// TIA Portal project "HW_2200220OffsetBodu_V18_V19" (V19)

(* hardware
DEVICE "ET 200SP station_1"  ET 200SP-Station
   slot 0: "IO-R3"  Rack  6ES5 710-8MAx1
   slot 0: "A6"  IM 155-6 PN ST  6ES7 155-6AU01-0BN0  V4.2
   slot 1: "15A2"  DI 16x24VDC ST  6ES7 131-6BH01-0BA0  V0.0
      slot 1: "15A2"  DI 16x24VDC ST
   slot 2: "15A3"  DI 16x24VDC ST  6ES7 131-6BH01-0BA0  V0.0
      slot 1: "15A3"  DI 16x24VDC ST
   slot 3: "15A4"  DI 16x24VDC ST  6ES7 131-6BH01-0BA0  V0.0
      slot 1: "15A4"  DI 16x24VDC ST
   slot 4: "15A5"  DQ 16x24VDC/0.5A ST  6ES7 132-6BH01-0BA0  V0.0
      slot 1: "15A5"  DQ 16x24VDC/0.5A ST
   slot 5: "15A6"  DQ 16x24VDC/0.5A ST  6ES7 132-6BH01-0BA0  V0.0
      slot 1: "15A6"  DQ 16x24VDC/0.5A ST
   slot 6: "15A7"  DQ 16x24VDC/0.5A ST  6ES7 132-6BH01-0BA0  V0.0
      slot 1: "15A7"  DQ 16x24VDC/0.5A ST
   slot 7: "15A8"  DQ 16x24VDC/0.5A ST  6ES7 132-6BH01-0BA0  V0.0
      slot 1: "15A8"  DQ 16x24VDC/0.5A ST
   slot 8: "15A9"  AI 4xU/I 2-wire ST  6ES7 134-6HD00-0BA1  V1.1
      slot 1: "15A9"  AI 4xU/I 2-wire ST
   slot 9: "15A10"  AQ 4xU/I ST  6ES7 135-6HD00-0BA1  V1.1
      slot 1: "15A10"  AQ 4xU/I ST
   slot 15: "Server module_1"  Server module  6ES7 193-6PA00-0AA0  V1.0
      slot 1: "Server module_1"  Server module
   slot 127: "PROFINET BusAdapter CU"  BA 2xRJ45  6ES7 193-6AR00-0AA0  V0.0
      slot 1: "Port_1"  X1 P1 R  6ES7 193-6AR00-0AA0  V0.0
      slot 2: "Port_2"  X1 P2 R  6ES7 193-6AR00-0AA0  V0.0
DEVICE "GSD device_7"  GSD.Device.PN
   slot 0: "Rack"  Rack  V1.0
   slot 0: "VI-13"  CPX Rev 30  TN 197330  V4.2.30
      slot 0: "CPX Rev 30"  CPX Rev 30
      slot 1: "PN-IO Interface"  PN-IO Interface
         slot 1: "Port 1"  Port 1
         slot 2: "Port 2"  Port 2
   slot 1: "FB33 PNIO Module_1"  FB33 PNIO Module  TN 548755, CPX-FB33, Code F33
      slot 0: "FB33 PNIO Module"  FB33 PNIO Module
   slot 2: "MPA1S VMPA1-FB-EMS-8 [8DO]_1"  MPA1S VMPA1-FB-EMS-8 [8DO]  TN 533360, VMPA1-FB-EMS-8, Code A
      slot 0: "MPA1S VMPA1-FB-EMS-8 [8DO]"  MPA1S VMPA1-FB-EMS-8 [8DO]
   slot 3: "MPA1S VMPA1-FB-EMS-8 [8DO]_2"  MPA1S VMPA1-FB-EMS-8 [8DO]  TN 533360, VMPA1-FB-EMS-8, Code A
      slot 0: "MPA1S VMPA1-FB-EMS-8 [8DO]"  MPA1S VMPA1-FB-EMS-8 [8DO]
   slot 4: "MPA1S VMPA1-FB-EMS-8 [8DO]_3"  MPA1S VMPA1-FB-EMS-8 [8DO]  TN 533360, VMPA1-FB-EMS-8, Code A
      slot 0: "MPA1S VMPA1-FB-EMS-8 [8DO]"  MPA1S VMPA1-FB-EMS-8 [8DO]
   slot 5: "MPA1S VMPA1-FB-EMS-8 [8DO]_4"  MPA1S VMPA1-FB-EMS-8 [8DO]  TN 533360, VMPA1-FB-EMS-8, Code A
      slot 0: "MPA1S VMPA1-FB-EMS-8 [8DO]"  MPA1S VMPA1-FB-EMS-8 [8DO]
   slot 6: "MPA1S VMPA1-FB-EMS-8 [8DO]_5"  MPA1S VMPA1-FB-EMS-8 [8DO]  TN 533360, VMPA1-FB-EMS-8, Code A
      slot 0: "MPA1S VMPA1-FB-EMS-8 [8DO]"  MPA1S VMPA1-FB-EMS-8 [8DO]
   slot 7: "MPA1S VMPA1-FB-EMS-8 [8DO]_6"  MPA1S VMPA1-FB-EMS-8 [8DO]  TN 533360, VMPA1-FB-EMS-8, Code A
      slot 0: "MPA1S VMPA1-FB-EMS-8 [8DO]"  MPA1S VMPA1-FB-EMS-8 [8DO]
   slot 8: "MPA1S VMPA1-FB-EMS-8 [8DO]_7"  MPA1S VMPA1-FB-EMS-8 [8DO]  TN 533360, VMPA1-FB-EMS-8, Code A
      slot 0: "MPA1S VMPA1-FB-EMS-8 [8DO]"  MPA1S VMPA1-FB-EMS-8 [8DO]
   slot 9: "MPA1S VMPA1-FB-EMS-8 [8DO]_8"  MPA1S VMPA1-FB-EMS-8 [8DO]  TN 533360, VMPA1-FB-EMS-8, Code A
      slot 0: "MPA1S VMPA1-FB-EMS-8 [8DO]"  MPA1S VMPA1-FB-EMS-8 [8DO]
DEVICE "Connection Box_1"  SCALANCE X-Station
   slot 0: "Connection Box"  Rail
   slot 0: "ConBox"  Connection Box advanced  6AV2 125-2AE23-0AX0  V5.2
DEVICE "GSD device_3"  GSD.Device.PN
   slot 0: "Rack"  Rack  V1.0
   slot 0: "AxisLinear"  CMMT-AS V1  CMMT-AS-...-PN
      slot 0: "CMMT-AS V1"  CMMT-AS V1
      slot 1: "PN-IO Interface"  PN-IO Interface
         slot 1: "Port 1"  Port 1
         slot 2: "Port 2"  Port 2
      slot 1: "DO SERVO_1"  DO SERVO
         slot 0: "Module Access Point"  Module Access Point
   slot 2: "Siemens telegram 111, PZD-12/12"  Siemens telegram 111, PZD-12/12
DEVICE "ET 200AL station_1"  ET 200AL-Station
   slot 0: "Rack_0"  Rack
   slot 0: "52K1"  IM 157-1 PN  6ES7 157-1AB00-0AB0  V1.0
      slot 1: "ET-Con_1"  ET-Con IM Sub-Sender
      slot 1: "ET-Con_2"  ET-Con IM Sub-Sender
   slot 1: "Rack_1"  Rack  6ES714x-xxxxx-0AA0
   slot 2: "Rack_2"  Rack  6ES714x-xxxxx-0AA0
   slot 2: "53AB1"  DI 8x24VDC 8xM8  6ES7 141-5BF00-0BA0  V1.0
      slot 1: "53AB1"  DI 8x24VDC 8xM8  6ES7 141-5BF00-0BA0
      slot 2: "ET-Connection receiver"  ET-Con Sub-Receiver
   slot 3: "54AB2"  DI 8x24VDC 8xM8  6ES7 141-5BF00-0BA0  V1.0
      slot 1: "54AB2"  DI 8x24VDC 8xM8  6ES7 141-5BF00-0BA0
   slot 4: "55AB3"  DI 8x24VDC 8xM8  6ES7 141-5BF00-0BA0  V1.0
      slot 1: "55AB3"  DI 8x24VDC 8xM8  6ES7 141-5BF00-0BA0
   slot 5: "56AB4"  DI 8x24VDC 8xM8  6ES7 141-5BF00-0BA0  V1.0
      slot 1: "56AB4"  DI 8x24VDC 8xM8  6ES7 141-5BF00-0BA0
   slot 6: "57AB5"  DI 8x24VDC 8xM8  6ES7 141-5BF00-0BA0  V1.0
      slot 1: "57AB5"  DI 8x24VDC 8xM8  6ES7 141-5BF00-0BA0
   slot 19: "58AB6"  AI 4xU/I/RTD 4xM12  6ES7 144-5KD00-0BA0  V1.0
      slot 1: "58AB6"  AI 4xU/I/RTD 4xM12  6ES7 144-5KD00-0BA0
      slot 2: "ET-Connection receiver"  ET-Con Sub-Receiver
   slot 20: "59AB7"  DI 8x24VDC 8xM8  6ES7 141-5BF00-0BA0  V1.0
      slot 1: "59AB7"  DI 8x24VDC 8xM8  6ES7 141-5BF00-0BA0
   slot 21: "59aAB7"  DI 8x24VDC 8xM8  6ES7 141-5BF00-0BA0  V1.0
      slot 1: "59aAB7"  DI 8x24VDC 8xM8  6ES7 141-5BF00-0BA0
   slot 22: "60AB8"  DI 8x24VDC 8xM8  6ES7 141-5BF00-0BA0  V1.0
      slot 1: "60AB8"  DI 8x24VDC 8xM8  6ES7 141-5BF00-0BA0
   slot 23: "61AB9"  DI 8x24VDC 8xM8  6ES7 141-5BF00-0BA0  V1.0
      slot 1: "61AB9"  DI 8x24VDC 8xM8  6ES7 141-5BF00-0BA0
   slot 24: "62AB10"  DI 8x24VDC 8xM8  6ES7 141-5BF00-0BA0  V1.0
      slot 1: "62AB10"  DI 8x24VDC 8xM8  6ES7 141-5BF00-0BA0
DEVICE "CVIC II R2 A"  GSD.Device.PN
   slot 0: "Rack"  Rack  V1.0
   slot 0: "Bash"  RT  ABCC-PRT  V1.11
      slot 0: "RT"  RT
      slot 1: "Interface"  Interface
         slot 1: "Port 1"  Port 1
   slot 1: "Input 1 byte_1"  Input 1 byte  ABCC-PRT  V1.0
      slot 0: "Input 1 byte"  Input 1 byte
   slot 2: "Input 1 byte_2"  Input 1 byte  ABCC-PRT  V1.0
      slot 0: "Input 1 byte"  Input 1 byte
   slot 3: "Input 2 word_1"  Input 2 word  ABCC-PRT  V1.0
      slot 0: "Input 2 word"  Input 2 word
   slot 4: "Input 1 word_1"  Input 1 word  ABCC-PRT  V1.0
      slot 0: "Input 1 word"  Input 1 word
   slot 5: "Input 2 word_2"  Input 2 word  ABCC-PRT  V1.0
      slot 0: "Input 2 word"  Input 2 word
   slot 6: "Input 1 word_2"  Input 1 word  ABCC-PRT  V1.0
      slot 0: "Input 1 word"  Input 1 word
   slot 7: "Output 1 byte_1"  Output 1 byte  ABCC-PRT  V1.0
      slot 0: "Output 1 byte"  Output 1 byte
   slot 8: "Output 1 byte_2"  Output 1 byte  ABCC-PRT  V1.0
      slot 0: "Output 1 byte"  Output 1 byte
DEVICE "CVIC II R2 A_1"  GSD.Device.PN
   slot 0: "Rack"  Rack  V1.0
   slot 0: "AEBDown"  RT  ABCC-PRT  V1.11
      slot 0: "RT"  RT
      slot 1: "Interface"  Interface
         slot 1: "Port 1"  Port 1
   slot 1: "Input 1 byte_1"  Input 1 byte  ABCC-PRT  V1.0
      slot 0: "Input 1 byte"  Input 1 byte
   slot 2: "Input 1 byte_2"  Input 1 byte  ABCC-PRT  V1.0
      slot 0: "Input 1 byte"  Input 1 byte
   slot 3: "Input 2 word_1"  Input 2 word  ABCC-PRT  V1.0
      slot 0: "Input 2 word"  Input 2 word
   slot 4: "Input 1 word_1"  Input 1 word  ABCC-PRT  V1.0
      slot 0: "Input 1 word"  Input 1 word
   slot 5: "Input 2 word_2"  Input 2 word  ABCC-PRT  V1.0
      slot 0: "Input 2 word"  Input 2 word
   slot 6: "Input 1 word_2"  Input 1 word  ABCC-PRT  V1.0
      slot 0: "Input 1 word"  Input 1 word
   slot 7: "Output 1 byte_1"  Output 1 byte  ABCC-PRT  V1.0
      slot 0: "Output 1 byte"  Output 1 byte
   slot 8: "Output 1 byte_2"  Output 1 byte  ABCC-PRT  V1.0
      slot 0: "Output 1 byte"  Output 1 byte
DEVICE "CVIC II R2 A_2"  GSD.Device.PN
   slot 0: "Rack"  Rack  V1.0
   slot 0: "AEBUp"  RT  ABCC-PRT  V1.11
      slot 0: "RT"  RT
      slot 1: "Interface"  Interface
         slot 1: "Port 1"  Port 1
   slot 1: "Input 1 byte_1"  Input 1 byte  ABCC-PRT  V1.0
      slot 0: "Input 1 byte"  Input 1 byte
   slot 2: "Input 1 byte_2"  Input 1 byte  ABCC-PRT  V1.0
      slot 0: "Input 1 byte"  Input 1 byte
   slot 3: "Input 2 word_1"  Input 2 word  ABCC-PRT  V1.0
      slot 0: "Input 2 word"  Input 2 word
   slot 4: "Input 1 word_1"  Input 1 word  ABCC-PRT  V1.0
      slot 0: "Input 1 word"  Input 1 word
   slot 5: "Input 2 word_2"  Input 2 word  ABCC-PRT  V1.0
      slot 0: "Input 2 word"  Input 2 word
   slot 6: "Input 1 word_2"  Input 1 word  ABCC-PRT  V1.0
      slot 0: "Input 1 word"  Input 1 word
   slot 7: "Output 1 byte_1"  Output 1 byte  ABCC-PRT  V1.0
      slot 0: "Output 1 byte"  Output 1 byte
   slot 8: "Output 1 byte_2"  Output 1 byte  ABCC-PRT  V1.0
      slot 0: "Output 1 byte"  Output 1 byte
DEVICE "CVIC II R2 A_3"  GSD.Device.PN
   slot 0: "Rack"  Rack  V1.0
   slot 0: "AETDown"  RT  ABCC-PRT  V1.11
      slot 0: "RT"  RT
      slot 1: "Interface"  Interface
         slot 1: "Port 1"  Port 1
   slot 1: "Input 1 byte_1"  Input 1 byte  ABCC-PRT  V1.0
      slot 0: "Input 1 byte"  Input 1 byte
   slot 2: "Input 1 byte_2"  Input 1 byte  ABCC-PRT  V1.0
      slot 0: "Input 1 byte"  Input 1 byte
   slot 3: "Input 2 word_1"  Input 2 word  ABCC-PRT  V1.0
      slot 0: "Input 2 word"  Input 2 word
   slot 4: "Input 1 word_1"  Input 1 word  ABCC-PRT  V1.0
      slot 0: "Input 1 word"  Input 1 word
   slot 5: "Input 2 word_2"  Input 2 word  ABCC-PRT  V1.0
      slot 0: "Input 2 word"  Input 2 word
   slot 6: "Input 1 word_2"  Input 1 word  ABCC-PRT  V1.0
      slot 0: "Input 1 word"  Input 1 word
   slot 7: "Output 1 byte_1"  Output 1 byte  ABCC-PRT  V1.0
      slot 0: "Output 1 byte"  Output 1 byte
   slot 8: "Output 1 byte_2"  Output 1 byte  ABCC-PRT  V1.0
      slot 0: "Output 1 byte"  Output 1 byte
DEVICE "CVIC II R2 A_4"  GSD.Device.PN
   slot 0: "Rack"  Rack  V1.0
   slot 0: "AETUp"  RT  ABCC-PRT  V1.11
      slot 0: "RT"  RT
      slot 1: "Interface"  Interface
         slot 1: "Port 1"  Port 1
   slot 1: "Input 1 byte_1"  Input 1 byte  ABCC-PRT  V1.0
      slot 0: "Input 1 byte"  Input 1 byte
   slot 2: "Input 1 byte_2"  Input 1 byte  ABCC-PRT  V1.0
      slot 0: "Input 1 byte"  Input 1 byte
   slot 3: "Input 2 word_1"  Input 2 word  ABCC-PRT  V1.0
      slot 0: "Input 2 word"  Input 2 word
   slot 4: "Input 1 word_1"  Input 1 word  ABCC-PRT  V1.0
      slot 0: "Input 1 word"  Input 1 word
   slot 5: "Input 2 word_2"  Input 2 word  ABCC-PRT  V1.0
      slot 0: "Input 2 word"  Input 2 word
   slot 6: "Input 1 word_2"  Input 1 word  ABCC-PRT  V1.0
      slot 0: "Input 1 word"  Input 1 word
   slot 7: "Output 1 byte_1"  Output 1 byte  ABCC-PRT  V1.0
      slot 0: "Output 1 byte"  Output 1 byte
   slot 8: "Output 1 byte_2"  Output 1 byte  ABCC-PRT  V1.0
      slot 0: "Output 1 byte"  Output 1 byte
DEVICE "GSD device_11"  GSD.Device.PN
   slot 0: "Rack"  Rack  V1.0
   slot 0: "GT2"  DL-PN1  DL-PN1  1.00
      slot 0: "DL-PN1"  DL-PN1  1.00
      slot 1: "Interface"  Interface
         slot 1: "Port 1"  Port 1
   slot 1: "DL-PN1_1"  DL-PN1
      slot 0: "DL-PN1 Device"  DL-PN1 Device
   slot 2: "B1"  GT2-***
      slot 0: "GT2-***"  GT2-***
   slot 3: "B2"  GT2-***
      slot 0: "GT2-***"  GT2-***
   slot 4: "B3"  GT2-***
      slot 0: "GT2-***"  GT2-***
   slot 5: "B4"  GT2-***
      slot 0: "GT2-***"  GT2-***
   slot 6: "B5"  GT2-***
      slot 0: "GT2-***"  GT2-***
   slot 7: "B6"  GT2-***
      slot 0: "GT2-***"  GT2-***
   slot 8: "B7"  GT2-***
      slot 0: "GT2-***"  GT2-***
   slot 9: "B8"  GT2-***
      slot 0: "GT2-***"  GT2-***
   slot 10: "B9"  GT2-***
      slot 0: "GT2-***"  GT2-***
DEVICE "GSD device_1"  GSD.Device.PN
   slot 0: "Rack"  Rack  V1.0
   slot 0: "CPX"  CPX-E-CEC V1  CPX-E-CEC-PN  V1.0.4
      slot 0: "CPX-E-CEC V1"  CPX-E-CEC V1
      slot 1: "PN-IO Interface"  PN-IO Interface
         slot 1: "Port 1"  Port 1
         slot 2: "Port 2"  Port 2
   slot 1: "CW_SW"  IO 4 byte
      slot 0: "IO 4 byte"  IO 4 byte
   slot 2: "CNC"  IO 32 byte
      slot 0: "IO 32 byte"  IO 32 byte
   slot 3: "PtP"  IO 16 byte
      slot 0: "IO 16 byte"  IO 16 byte
   slot 4: "Error"  IO 32 byte
      slot 0: "IO 32 byte"  IO 32 byte
DEVICE "GSD device_2"  GSD.Device.PN
   slot 0: "Rack"  Rack  V1.0
   slot 0: "Reader"  SR-1000X  SR-1000X  1.0
      slot 0: "SR-1000X"  SR-1000X  1.0
      slot 1: "Interface"  Interface
         slot 1: "Port 1"  Port 1
   slot 1: "Handshake and General Error Status Bits_1"  Handshake and General Error Status Bits
      slot 0: "Handshake and General Error Status Bits"  Handshake and General Error Status Bits
   slot 2: "BUSY Status Bits_1"  BUSY Status Bits
      slot 0: "BUSY Status Bits"  BUSY Status Bits
   slot 3: "Completion Status Bits_1"  Completion Status Bits
      slot 0: "Completion Status Bits"  Completion Status Bits
   slot 4: "Error Status Bits_1"  Error Status Bits
      slot 0: "Error Status Bits"  Error Status Bits
   slot 5: "Terminal Status Bits_1"  Terminal Status Bits
      slot 0: "Terminal Status Bits"  Terminal Status Bits
   slot 6: "Unstable Read Status Bits_1"  Unstable Read Status Bits
      slot 0: "Unstable Read Status Bits"  Unstable Read Status Bits
   slot 7: "Matching Level and Total Evaluation Grade Status_1"  Matching Level and Total Evaluation Grade Status
      slot 0: "Matching Level and Total Evaluation Grade Status"  Matching Level and Total Evaluation Grade Status
   slot 8: "Operation Result Status_1"  Operation Result Status
      slot 0: "Operation Result Status"  Operation Result Status
   slot 9: "Read Data 128Byte_1"  Read Data 128Byte
      slot 0: "Read Data 128Byte"  Read Data 128Byte
   slot 10: "Latch and Error Clear Control Bits_1"  Latch and Error Clear Control Bits
      slot 0: "Latch and Error Clear Control Bits"  Latch and Error Clear Control Bits
   slot 11: "Operation instruction Control Bits_1"  Operation instruction Control Bits
      slot 0: "Operation instruction Control Bits"  Operation instruction Control Bits
   slot 12: "Completion Clear Control Bits_1"  Completion Clear Control Bits
      slot 0: "Completion Clear Control Bits"  Completion Clear Control Bits
   slot 13: "Parameter Bank Number_1"  Parameter Bank Number
      slot 0: "Parameter Bank Number"  Parameter Bank Number
   slot 14: "User Data 128Byte_1"  User Data 128Byte
      slot 0: "User Data 128Byte"  User Data 128Byte
DEVICE "S71500/ET200MP station_1"  S7-1500 station
   slot 0: "Rail_0"  Rack  6ES7 590-1***0-0AA0
   slot 1: "A5"  CPU 1516F-3 PN/DP  6ES7 516-3FN02-0AB0  V2.9
      slot 3: "CPU display_1"  6ES7591-1BA00-0AA0
      slot 32768: "PROFINET interface_1"  X1
         slot 32769: "Port_1"  X1 P1
         slot 32770: "Port_2"  X1 P2
      slot 33024: "PROFINET interface_2"  X2
         slot 33025: "Port_1"  X2 P1
      slot 33280: "DP interface_1"  X3
      slot 34817: "Virtual CP interface port_1"  Virtual CP interface port  Virtual CP interface port
*)

// ===== PLC "A5"  CPU 1516F-3 PN/DP =====

VAR_GLOBAL   // PLC tag table "Default tag table"
   "Clock_Byte" AT %MB0 : Byte;
   "Clock_10Hz" AT %M0.0 : Bool;
   "Clock_5Hz" AT %M0.1 : Bool;
   "Clock_2.5Hz" AT %M0.2 : Bool;
   "Clock_2Hz" AT %M0.3 : Bool;
   "Clock_1.25Hz" AT %M0.4 : Bool;
   "Clock_1Hz" AT %M0.5 : Bool;
   "Clock_0.625Hz" AT %M0.6 : Bool;
   "Clock_0.5Hz" AT %M0.7 : Bool;
   "System_Byte" AT %MB1 : Byte;
   "FirstScan" AT %M1.0 : Bool;
   "DiagStatusUpdate" AT %M1.1 : Bool;
   "AlwaysTRUE" AT %M1.2 : Bool;
   "AlwaysFALSE" AT %M1.3 : Bool;
END_VAR

DATA_BLOCK "Main_Safety_RTG1_DB"   // DB1, F_DB
{ S7_Optimized_Access := 'TRUE' }
NAME : FUSI
VERSION : 0.1
// stored: InstanceOfName Main_Safety_RTG1
"Main_Safety_RTG1"
BEGIN
END_DATA_BLOCK

FUNCTION_BLOCK "Main_Safety_RTG1"   // FB1, F_FBD
{ S7_Optimized_Access := 'TRUE' }
BEGIN
END_FUNCTION_BLOCK

ORGANIZATION_BLOCK "Main"   // OB1, LAD, ProgramCycle
TITLE = "Main Program Sweep (Cycle)"
{ S7_Optimized_Access := 'TRUE' }
VERSION : 0.1
   VAR_INPUT
      Initial_Call : Bool;   // Initial call of this OB
      Remanence : Bool;   // =True, if remanent data are available
   END_VAR
BEGIN
END_ORGANIZATION_BLOCK